PROGRAM MAIN
VAR
	bActivateMotion 	: BOOL;
	fVelRef 			: LREAL;
	fPosRef 			: LREAL;
	fPosMeas 			: LREAL;
	fPres1Meas			: LREAL;
	fPres2Meas			: LREAL;
END_VAR

P_Commissioning();
P_ControlBox();
P_CraneControl();

G_Simulator.bSimulatorOn := bActivateMotion;
fPosMeas := G_Simulator.fBoomAngle;
G_Commissioning.stMotionReferenceGeneratorSettings.fPositionSetpoint_ms := fVelRef;
G_Commissioning.stMotionReferenceGeneratorSettings.fHoldPositionTime_s := 1000.0;
fPres1Meas := G_Simulator.fPistonSidePressure;
fPres2Meas := G_Simulator.fRodSidePressure;

END_PROGRAM

(* stored: Version 1.1.0.1, ProductVersion 3.1.4024.12
   POU MAIN: Id {710c49b1-6c28-4dfa-b3ee-ba840c2a49f8}, SpecialFunc None *)
